FUNCTION_BLOCK LIMIT_REAL (* See LIMIT_ANY *)
  (* Standard: 61131-3 *)
  (* Version 0.0, 2004-12-15, JHC, Rockwell Automation, Converted from SRC format. *)
  (* Compiler header: package fb.rt.plc.select; *)
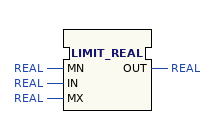
  VAR_INPUT
    MN : REAL;
    IN : REAL;
    MX : REAL;
  END_VAR
  VAR_OUTPUT
    OUT : REAL;
  END_VAR
END_FUNCTION_BLOCK
